// TwinCAT 3 PLC project plc1
// ProgramVersion: 3.1.4024.0
// libraries:
//   Tc2_Standard, * (Beckhoff Automation GmbH)
//   Tc2_System, * (Beckhoff Automation GmbH)
//   Tc3_Module, * (Beckhoff Automation GmbH)
// project tree:
//   / PlcTask.TcTTO
//   POUs/ MAIN.TcPOU
// real-time tasks:
//   TASK PlcTask: cycle T#10ms, priority 20, ADS port 350
// I/O:
//   DEVICE Dispositivo 1 (EtherCAT Automation Protocol), AmsNetId 5.135.111.161.2.1
//   DEVICE Dispositivo 2 (EtherCAT Automation Protocol), AmsNetId 5.135.111.161.3.1
//   DEVICE Dispositivo 3 (COM Port)
//   DEVICE Dispositivo 4 (EtherCAT), AmsNetId 5.135.111.161.5.1
//     Terminal 1 (EK1200) [EK1200-5000 EtherCAT Power supply (2A E-Bus)]
//       Terminal 2 (EL1002) [EL1002 2Ch. Dig. Input 24V, 3ms]
//       Terminal 3 (EL2002) [EL2002 2Ch. Dig. Output 24V, 0.5A]
//       Terminal 4 (EL9011) [EL9011 End Terminal]

CONFIGURATION plc1
    RESOURCE PLC ON TwinCAT3
        TASK PlcTask(INTERVAL := T#10ms, PRIORITY := 20);
        PROGRAM MAIN WITH PlcTask : MAIN;
    END_RESOURCE
END_CONFIGURATION

// ---- POUs/MAIN.TcPOU
PROGRAM MAIN
VAR
END_VAR

END_PROGRAM
